// Mitsubishi GX Works2 project: 0708-산술실수   PLC: Q02/Q02H

PROGRAM MAIN
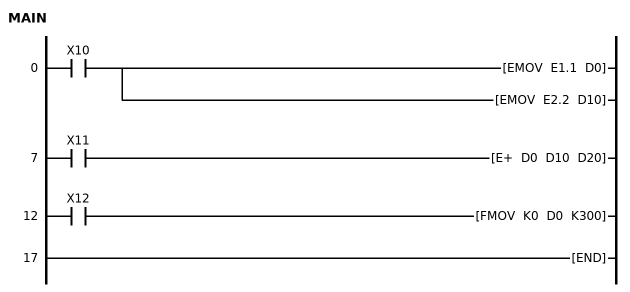
0     LD      X10
      EMOV    E1.1 D0
      EMOV    E2.2 D10
7     LD      X11
      E+      D0 D10 D20
12    LD      X12
      FMOV    K0 D0 K300
17    END
END_PROGRAM
